INTERFACE I_RpcMiddlewareConfig

PROPERTY PUBLIC ContentType_Json : T_MAXSTRING
GET
END_GET
SET
END_SET
END_PROPERTY

METHOD PUBLIC TryGetAcceptResponseFormatFromRequest : BOOL
VAR_INPUT
	Request : I_Request;
	Destination : ANY;
END_VAR
END_METHOD

METHOD PUBLIC TryGetContentTypeFromRequest : BOOL
VAR_INPUT
	Request : I_Request;
	Destination : ANY;
END_VAR
END_METHOD

METHOD PUBLIC TryGetMethodNameFromRequest : BOOL
VAR_INPUT
	Request : I_Request;
	Destination : ANY;
END_VAR
END_METHOD

METHOD PUBLIC TryGetTypeFromRequest : BOOL
VAR_INPUT
	Request : I_Request;
	Destination : ANY;
END_VAR
END_METHOD

END_INTERFACE

(* stored: Version 1.1.0.1, ProductVersion 3.1.4024.12
   Itf I_RpcMiddlewareConfig: Id {f56a132e-091f-4d11-8291-aa2e1482fb04}
   Property ContentType_Json: Id {1a976427-ee75-4904-bad1-149db0babafa}
   Get Get: Id {33ad120c-bf8e-4d4a-a6a6-33330b2a4f67}
   Set Set: Id {d8798428-7853-49b1-bf78-53ea471c9bcb}
   Method TryGetAcceptResponseFormatFromRequest: Id {e0a58c28-b602-48b9-a496-db1f0b89979a}
   Method TryGetContentTypeFromRequest: Id {94705d98-85e5-457d-8454-37b8f95e13cf}
   Method TryGetMethodNameFromRequest: Id {a65d65b3-7d7f-4720-adda-86351a60f618}
   Method TryGetTypeFromRequest: Id {cb572c29-36dc-446c-b007-c1aec0312c5f} *)
